{attribute 'GeneratedUsingTerminal: EL7342-0000-0022'}
{attribute addProperty BoxType "EL7342-0000-0022"}
{attribute addProperty Id "Enable_latch_extern_on_positive_edgeBOOL1Set_counterBOOL1Enable_latch_extern_on_negative_edgeBOOL1"}
{attribute addProperty CRC "4052334391"}
{attribute addProperty Size "3"}
TYPE Control_F189B737 :
STRUCT
	{attribute addProperty Name "Enable_latch_extern_on_positive_edge"}
	Enable_latch_extern_on_positive_edge : BOOL;
	{attribute addProperty Name "Set_counter"}
	Set_counter : BOOL;
	{attribute addProperty Name "Enable_latch_extern_on_negative_edge"}
	Enable_latch_extern_on_negative_edge : BOOL;
END_STRUCT
END_TYPE

(* stored: Version 1.2.0.0
   DUT Control_F189B737: Id {ace95f7f-cdfb-4cd8-b040-2358a76221c9} *)
